{attribute 'GeneratedUsingTerminal: KL1501-0001'}
{attribute addProperty BoxType "KL1501-0001"}
{attribute addProperty Description ""}
{attribute addProperty Physics ""}
{attribute addProperty Id "Channel_1AT %Q*Channel_B5275D8E0"}
{attribute addProperty CRC "1658610108"}
{attribute addProperty Size "0"}
TYPE KL_62DC61BC :
STRUCT
	{attribute addProperty Name "Channel_1"}
	Channel_1 : Channel_B5275D8E;
END_STRUCT
END_TYPE

(* stored: Version 1.2.0.0, ProductVersion 3.1.4024.9
   DUT KL_62DC61BC: Id {7085cf7f-b66e-45b0-8687-ba570c9a2b31} *)
